# EPICS alarm handler configuration: css_share/detectors/SVT/alh/SVT.R3.alhConfig
GROUP NULL R3
INCLUDE R3 SVT.R3.S1.alhConfig
INCLUDE R3 SVT.R3.S2.alhConfig
INCLUDE R3 SVT.R3.S3.alhConfig
INCLUDE R3 SVT.R3.S4.alhConfig
INCLUDE R3 SVT.R3.S5.alhConfig
INCLUDE R3 SVT.R3.S6.alhConfig
INCLUDE R3 SVT.R3.S7.alhConfig
INCLUDE R3 SVT.R3.S8.alhConfig
INCLUDE R3 SVT.R3.S9.alhConfig
INCLUDE R3 SVT.R3.S10.alhConfig
INCLUDE R3 SVT.R3.S11.alhConfig
INCLUDE R3 SVT.R3.S12.alhConfig
INCLUDE R3 SVT.R3.S13.alhConfig
INCLUDE R3 SVT.R3.S14.alhConfig
INCLUDE R3 SVT.R3.S15.alhConfig
INCLUDE R3 SVT.R3.S16.alhConfig
INCLUDE R3 SVT.R3.S17.alhConfig
INCLUDE R3 SVT.R3.S18.alhConfig
